Fanuc KAREL source: kt00514.KL

PROGRAM KT00514
%STACKSIZE=65535
%PRIORITY=65535
%NOLOCKGROUP
VAR
P1 : XYZWPREXT
P2 : POSITION
OUT : POSITION
BEGIN
P1.X=1.0
-- UNRESOLVED_PC line 9 opcodes [49 7E 49 60 4A] marker_code=20
END KT00514
